{attribute 'qualified_only'}
{attribute 'strict'}
TYPE TopMaterialsEnum :
(
	//CARDBOARD
	CAR20S, CAR20M, CAR20L, CAR28S, CAR28M, CAR28L, //base (flat)
	
	//CHIPBOARD
	CIP18, CIP54,
	
	//WOOD BUNK
	WDT20, WDT22, WDT28, //top
	WDW20, WDW22, //special top (wide)
	
	size //number of materials
);
END_TYPE

(* stored: Version 1.1.0.1, ProductVersion 3.1.4024.11
   EnumerationTextList TopMaterialsEnum: Id {a8461138-96ed-4d25-a62c-024915123e2a} *)
